// TIA Portal V18 export
DATA_BLOCK "LCCF_EnetScanner_DB"   // DB4
// stored: InstanceOfName LCCF_EnetScanner, InstanceOfType FB
"LCCF_EnetScanner"
   // VAR_INPUT
   //    enable : Bool;
   //    interface { ExternalWritable := 'False'} : HW_INTERFACE;
   // END_VAR
   // VAR_OUTPUT
   //    valid { ExternalWritable := 'False'} : Bool;
   //    busy { ExternalWritable := 'False'} : Bool;
   //    error { ExternalWritable := 'False'} : Bool;
   //    isActive { ExternalWritable := 'False'} : Bool;
   //    status { ExternalWritable := 'False'} : Word;
   //    diagnostics { ExternalWritable := 'False'} : "LCCF_typeDiagnostics";
   // END_VAR
   // VAR_IN_OUT
   //    adapters : Array[*] of "LCCF_typeEnetAdaptConfig";
   //    data : Array[*] of "LCCF_typeEnetAdaptData";
   // END_VAR
   // VAR
   //    statEnableOld { ExternalAccessible := 'False'; ExternalVisible := 'False'; ExternalWritable := 'False'} : Bool;
   //    statValid { ExternalAccessible := 'False'; ExternalVisible := 'False'; ExternalWritable := 'False'} : Bool;
   //    statBusy { ExternalAccessible := 'False'; ExternalVisible := 'False'; ExternalWritable := 'False'} : Bool;
   //    statError { ExternalAccessible := 'False'; ExternalVisible := 'False'; ExternalWritable := 'False'} : Bool;
   //    statDataExchange { ExternalAccessible := 'False'; ExternalVisible := 'False'; ExternalWritable := 'False'} : Bool;
   //    statErrorUserCleared { ExternalAccessible := 'False'; ExternalVisible := 'False'; ExternalWritable := 'False'} : Bool;
   //    statErrorAutoCleared { ExternalAccessible := 'False'; ExternalVisible := 'False'; ExternalWritable := 'False'} : Bool;
   //    statDiagnostic { ExternalAccessible := 'False'; ExternalVisible := 'False'; ExternalWritable := 'False'} : "LCCF_typeDiagnostics";
   //    statEmptyDiagnostics { ExternalAccessible := 'False'; ExternalVisible := 'False'; ExternalWritable := 'False'} : "LCCF_typeDiagnostics";
   //    statMachineState { ExternalAccessible := 'False'; ExternalVisible := 'False'; ExternalWritable := 'False'} : DInt;
   //    statDisablingCompleted { ExternalAccessible := 'False'; ExternalVisible := 'False'; ExternalWritable := 'False'} : Bool;
   //    statWaitForInputUpdate { ExternalAccessible := 'False'; ExternalVisible := 'False'; ExternalWritable := 'False'} : Bool;
   //    statRequestLength { ExternalAccessible := 'False'; ExternalVisible := 'False'; ExternalWritable := 'False'} : UInt;
   //    statItemNumber { ExternalAccessible := 'False'; ExternalVisible := 'False'; ExternalWritable := 'False'} : UInt;
   //    statItemDataIndex { ExternalAccessible := 'False'; ExternalVisible := 'False'; ExternalWritable := 'False'} : UInt;
   //    statOwnContext { ExternalAccessible := 'False'; ExternalVisible := 'False'; ExternalWritable := 'False'} : Array[0..7] of USInt;
   //    instReadPnDevInterface { ExternalAccessible := 'False'; ExternalVisible := 'False'; ExternalWritable := 'False'; S7_SetPoint := 'True'} : RDREC;
   //    instDisconnect { ExternalAccessible := 'False'; ExternalVisible := 'False'; ExternalWritable := 'False'; S7_SetPoint := 'True'} : Array[0..15] of TDISCON;
   //    instConnect { ExternalAccessible := 'False'; ExternalVisible := 'False'; ExternalWritable := 'False'; S7_SetPoint := 'True'} : Array[0..15] of TCON;
   //    instSendManage { ExternalAccessible := 'False'; ExternalVisible := 'False'; ExternalWritable := 'False'; S7_SetPoint := 'True'} : Array[0..15] of TSEND;
   //    instReceiveManage { ExternalAccessible := 'False'; ExternalVisible := 'False'; ExternalWritable := 'False'; S7_SetPoint := 'True'} : Array[0..15] of TRCV;
   //    instSetupIO { ExternalAccessible := 'False'; ExternalVisible := 'False'; ExternalWritable := 'False'; S7_SetPoint := 'True'} : TCON;
   //    instResetIO { ExternalAccessible := 'False'; ExternalVisible := 'False'; ExternalWritable := 'False'; S7_SetPoint := 'True'} : TDISCON;
   //    instSendOutputs { ExternalAccessible := 'False'; ExternalVisible := 'False'; ExternalWritable := 'False'; S7_SetPoint := 'True'} : TUSEND;
   //    instRecvInputs { ExternalAccessible := 'False'; ExternalVisible := 'False'; ExternalWritable := 'False'; S7_SetPoint := 'True'} : TURCV;
   //    statUpdateQueue { ExternalAccessible := 'False'; ExternalVisible := 'False'; ExternalWritable := 'False'} : Struct
   //       requests : Array[0..15] of Bool;
   //       isProcessing : Array[0..15] of Bool;
   //       requestWarning : Array[0..15] of Bool;
   //    END_STRUCT;
   //    statAdapters { ExternalAccessible := 'False'; ExternalVisible := 'False'; ExternalWritable := 'False'} : Array[0..15] of Struct
   //       machineState : DInt;
   //       manageConnection { S7_SetPoint := 'True'} : TCON_IP_v4;
   //       ioRemotePort : UInt;
   //       instMgmtWatchdog { S7_SetPoint := 'True'} : IEC_TIMER;
   //       instTargetOrgWatchdog { S7_SetPoint := 'True'} : IEC_TIMER;
   //       instUpdateOutTrigger { S7_SetPoint := 'True'} : IEC_TIMER;
   //       instSettleTimer { S7_SetPoint := 'True'} : IEC_TIMER;
   //       instUpdateCfgTrigger { S7_SetPoint := 'True'} : IEC_TIMER;
   //       request : Struct
   //          header : Struct
   //             command : UInt;
   //             length : UInt;
   //             session : UDInt;
   //             status : UDInt;
   //             context : Array[0..7] of USInt;
   //             options : UDInt;
   //          END_STRUCT;
   //          data : Array[0..511] of USInt;
   //       END_STRUCT;
   //       response : Struct
   //          header : Struct
   //             command : UInt;
   //             length : UInt;
   //             session : UDInt;
   //             status : UDInt;
   //             context : Array[0..7] of USInt;
   //             options : UDInt;
   //          END_STRUCT;
   //          data : Array[0..511] of USInt;
   //       END_STRUCT;
   //       identity : Struct
   //          vendorID : UInt;
   //          deviceType : UInt;
   //          productCode : UInt;
   //          revision : Array[0..1] of USInt;
   //          serialNumber : UDInt;
   //          productName : String[64];
   //       END_STRUCT;
   //       statistics : Struct
   //          sendOctets : UDInt;
   //          recvdOctets : UDInt;
   //          inputApi : Struct
   //             start : LReal;
   //             stop : LReal;
   //             meter : LReal;
   //             maxInterval : LReal;
   //          END_STRUCT;
   //          outputApi : Struct
   //             start : LReal;
   //             stop : LReal;
   //             meter : LReal;
   //             maxInterval : LReal;
   //          END_STRUCT;
   //       END_STRUCT;
   //       mgmtTimeOut : Time;
   //       targetOrgTimeOut { S7_SetPoint := 'True'} : Time;
   //       orgTargetUpdateTime : Time;
   //       contedSeqNum : UInt;
   //       seqedAddrSeqNum : UDInt;
   //       watchDogErrorCounter : Int;
   //       serviceCapability : Word;
   //       sessionIdentifier : UDInt;
   //       targetOrgIdentifier : DWord;
   //       targetOrgInLength : UInt;
   //       orgTargetIdentifier : DWord;
   //       orgTargetOutLength : UInt;
   //       configOutLength : UInt;
   //       mgmtWatchdogGo : Bool;
   //       watchDogGo : Bool;
   //       updateOutputGo : Bool;
   //       updateConfigGo : Bool;
   //       settleConnectGo : Bool;
   //       updateConfig : Bool;
   //       isSettled : Bool;
   //       isEnabled : Bool;
   //       isInExchange : Bool;
   //       hasShutDown : Bool;
   //       isShuttingDown : Bool;
   //    END_STRUCT;
   //    statScanner { ExternalAccessible := 'False'; ExternalVisible := 'False'; ExternalWritable := 'False'} : Struct
   //       pnDevInterfaceData : Struct
   //          header : Struct
   //             recordType : UInt;
   //             recordLength : UInt;
   //             recordVersionMajor : USInt;
   //             recordVersionMinor : USInt;
   //          END_STRUCT;
   //          data : Array[0..255] of USInt;
   //       END_STRUCT;
   //       ownMacAddress : Array[0..5] of Byte;
   //       ownIpAddress { S7_SetPoint := 'True'} : IP_V4;
   //       activeAdapters { S7_SetPoint := 'True'} : Array[0..15] of Bool;
   //       ioConnection { S7_SetPoint := 'True'} : TCON_IP_v4;
   //       ioSendAddr { S7_SetPoint := 'True'} : TADDR_Param;
   //       ioRecvAddr { S7_SetPoint := 'True'} : TADDR_Param;
   //       instSettleTimer { S7_SetPoint := 'True'} : IEC_TIMER;
   //       settleConnectGo { S7_SetPoint := 'True'} : Bool;
   //    END_STRUCT;
   //    statOutputBuffer { ExternalAccessible := 'False'; ExternalVisible := 'False'; ExternalWritable := 'False'} : Struct
   //       itemCount : UInt;
   //       sequencedAddressItem : Struct
   //          typeIdentifier : UInt;
   //          length : UInt;
   //          connectionIdentifier : DWord;
   //          sequenceNumber : UDInt;
   //       END_STRUCT;
   //       connectedDataItem : Struct
   //          typeIdentifier : UInt;
   //          length : UInt;
   //          sequenceNumber : UInt;
   //          runIdleHeader : DWord;
   //          data : Array[0..497] of USInt;
   //       END_STRUCT;
   //    END_STRUCT;
   //    statInputBuffer { ExternalAccessible := 'False'; ExternalVisible := 'False'; ExternalWritable := 'False'} : Struct
   //       itemCount : UInt;
   //       sequencedAddressItem : Struct
   //          typeIdentifier : UInt;
   //          length : UInt;
   //          connectionIdentifier : DWord;
   //          sequenceNumber : UDInt;
   //       END_STRUCT;
   //       connectedDataItem : Struct
   //          typeIdentifier : UInt;
   //          length : UInt;
   //          sequenceNumber : UInt;
   //          data : Array[0..501] of USInt;
   //       END_STRUCT;
   //    END_STRUCT;
   //    statRandomNumGenerator { ExternalAccessible := 'False'; ExternalVisible := 'False'; ExternalWritable := 'False'} : Struct
   //       squared : DInt;
   //       weyl : DInt;
   //       value : UInt;
   //    END_STRUCT;
   //    statRuntimeInfo { ExternalAccessible := 'False'; ExternalVisible := 'False'; ExternalWritable := 'False'} : Struct
   //       start : LReal;
   //       stop : LReal;
   //       meter : LReal;
   //       maxInterval : LReal;
   //    END_STRUCT;
   //    statOutputLength { ExternalAccessible := 'False'; ExternalVisible := 'False'; ExternalWritable := 'False'} : UDInt;
   //    statOutUpdateTriggerGo { ExternalAccessible := 'False'; ExternalVisible := 'False'; ExternalWritable := 'False'} : Bool;
   //    statInUpdateWatchDogGo { ExternalAccessible := 'False'; ExternalVisible := 'False'; ExternalWritable := 'False'} : Bool;
   //    statInputIsUsint { ExternalAccessible := 'False'; ExternalVisible := 'False'; ExternalWritable := 'False'} : Bool;
   //    statInputIsUint { ExternalAccessible := 'False'; ExternalVisible := 'False'; ExternalWritable := 'False'} : Bool;
   //    statInputIsUdint { ExternalAccessible := 'False'; ExternalVisible := 'False'; ExternalWritable := 'False'} : Bool;
   //    statOutputIsUsint { ExternalAccessible := 'False'; ExternalVisible := 'False'; ExternalWritable := 'False'} : Bool;
   //    statOutputIsUint { ExternalAccessible := 'False'; ExternalVisible := 'False'; ExternalWritable := 'False'} : Bool;
   //    statOutputIsUdint { ExternalAccessible := 'False'; ExternalVisible := 'False'; ExternalWritable := 'False'} : Bool;
   //    statParamedOutBufferSize { ExternalAccessible := 'False'; ExternalVisible := 'False'; ExternalWritable := 'False'} : UInt;
   //    statParamedInBufferSize { ExternalAccessible := 'False'; ExternalVisible := 'False'; ExternalWritable := 'False'} : UInt;
   //    statRemainingData { ExternalAccessible := 'False'; ExternalVisible := 'False'; ExternalWritable := 'False'} : UInt;
   //    statBaseMacIndex { ExternalAccessible := 'False'; ExternalVisible := 'False'; ExternalWritable := 'False'} : Int;
   //    statTimeOut { ExternalAccessible := 'False'; ExternalVisible := 'False'; ExternalWritable := 'False'} : UInt;
   //    statReqPackInterval { ExternalAccessible := 'False'; ExternalVisible := 'False'; ExternalWritable := 'False'} : DInt;
   //    statConnectionParams { ExternalAccessible := 'False'; ExternalVisible := 'False'; ExternalWritable := 'False'} : Word;
   //    statItemCount { ExternalAccessible := 'False'; ExternalVisible := 'False'; ExternalWritable := 'False'} : UInt;
   //    statActItemIdentifier { ExternalAccessible := 'False'; ExternalVisible := 'False'; ExternalWritable := 'False'} : UInt;
   //    statActItemLength { ExternalAccessible := 'False'; ExternalVisible := 'False'; ExternalWritable := 'False'} : UInt;
   //    statCpfItemStartIndex { ExternalAccessible := 'False'; ExternalVisible := 'False'; ExternalWritable := 'False'} : UInt;
   //    statMoveOutputResult { ExternalAccessible := 'False'; ExternalVisible := 'False'; ExternalWritable := 'False'} : Int;
   //    statAdaptNameLength { ExternalAccessible := 'False'; ExternalVisible := 'False'; ExternalWritable := 'False'} : Int;
   //    statAdaptNameIndex { ExternalAccessible := 'False'; ExternalVisible := 'False'; ExternalWritable := 'False'} : Int;
   //    statMoveOutputIndex { ExternalAccessible := 'False'; ExternalVisible := 'False'; ExternalWritable := 'False'} : UInt;
   //    statOutSwapBufferUint { ExternalAccessible := 'False'; ExternalVisible := 'False'; ExternalWritable := 'False'} : UInt;
   //    statOutSwapBufferUdint { ExternalAccessible := 'False'; ExternalVisible := 'False'; ExternalWritable := 'False'} : UDInt;
   //    statAdaptNameLastIndex { ExternalAccessible := 'False'; ExternalVisible := 'False'; ExternalWritable := 'False'} : Int;
   //    statAdaptNameStartIndex { ExternalAccessible := 'False'; ExternalVisible := 'False'; ExternalWritable := 'False'} : Int;
   //    statProtocolVersion { ExternalAccessible := 'False'; ExternalVisible := 'False'; ExternalWritable := 'False'} : Word;
   //    statConfiguredAdapters { ExternalAccessible := 'False'; ExternalVisible := 'False'; ExternalWritable := 'False'} : DInt;
   //    statConfiguredAdaptersLow { ExternalAccessible := 'False'; ExternalVisible := 'False'; ExternalWritable := 'False'} : DInt;
   //    statConfiguredDataAreas { ExternalAccessible := 'False'; ExternalVisible := 'False'; ExternalWritable := 'False'} : DInt;
   //    statConfiguredDataAreasLow { ExternalAccessible := 'False'; ExternalVisible := 'False'; ExternalWritable := 'False'} : DInt;
   // END_VAR
BEGIN
END_DATA_BLOCK
